Universal Robots PolyScope program: UR_con_pick.urp

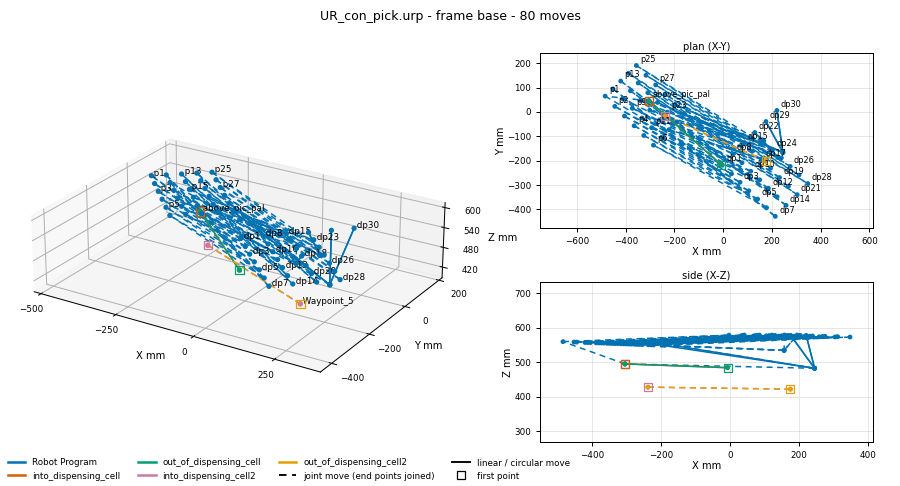
[picture p0: tool path of UR_con_pick.urp in frame base, 80 of 84 moves have a stored position in this frame; points joined in program order, loops and branches not executed]
Program UR_con_pick (installation=koniku1 directory=/programs/usbdisk createdIn=5.8.2.10297 lastSavedIn=5.8.2.10297 robotSerialNumber=20185300086)
Calibrated DH parameters: a=[0, -0.24355, -0.2132, 0, 0, 0]; d=[0.15185, 0, 0, 0.13105, 0.08535, 0.0921]; alpha=[1.570796, 0, 0, 1.570796, -1.570796, 0]; deltaTheta=[0, 0, 0, 0, 0, 0]
BeforeStart
  URCap Gripper Activate (Robotiq_Grippers, Robotiq Inc.) dataModel(ResetAndActivateKey=false)
  URCap Gripper (Robotiq_Grippers, Robotiq Inc.) dataModel(position=5.88235294117647, force=0.0, speed=100.0, positionInDouble=5.88235294117647, forceInDouble=0.0, speedInDouble=100.0, slaveIds=[9], blocking=true)
Robot Program (runOnlyOnce=false)
  Set DigitalOutput pin=digital_out[4]; digitalValue=0
  Set DigitalOutput pin=digital_out[5]; digitalValue=0
  Set DigitalOutput pin=digital_out[6]; digitalValue=1
  Wait DigitalInput pin=digital_in[0]; digitalValue=1
  Wait Sleep waitTime=2
  Set DigitalOutput pin=digital_out[4]; digitalValue=1
  SuppressedNode
    Call into_dispensing_cell
  Set DigitalOutput pin=digital_out[6]; digitalValue=0
  SuppressedNode
    Wait Sleep waitTime=4
  SuppressedNode
    Set DigitalOutput pin=digital_out[4]; digitalValue=0
  SuppressedNode
    Call out_of_dispensing_cell
  SuppressedNode
    URCap Palletizing (pallet-impl, Universal Robots) dataModel(palletFeature=Base, isPalletizing=true, Variable(key=globalCountingVariable, variable(name=Pallet_1_cnt, initializeExpression=1)), Variable(key=layerNumberVariable, variable(name=Pallet_1_lno, initializeExpression=1)), Variable(key=layerCountingVariable, variable(name=Pallet_1_lct, initializeExpression=1)), Variable(key=handleSeparatorVariable, variable(name=Pallet_1_sep, initializeExpression=False)), Variable(key=totalCountVariable, variable(name=Pallet_1_tct, initializeExpression=1)), Variable(key=name, variable(name=Pallet_pick)), Length(key=objectHeight value=0.007 unit=M), Variable(key=referencePoint, variable(featureName=referencePoint)), Variable(key=separatorPoint, variable(featureName=separatorPoint))); state(isChildrenLocked=true)
      URCap Patterns (pallet-impl, Universal Robots) state(isChildrenLocked=true)
        URCap Pattern (pallet-impl, Universal Robots) dataModel(UUID=97f9e36b-b9de-4589-9d53-87cbb1149383, patternType=GRID, rows=6, columns=5, Variable(key=nameVariable, variable(name=Grid_Pattern_1))); state(isChildrenLocked=true)
          URCap Item (pallet-impl, Universal Robots) dataModel(UUID=9fdc5ce5-b6e0-4f8b-9b1e-b639d3105400, patternType=GRID, index=0, calibrationDeltaTheta=[0.0, 0.0, 0.0, 0.0, 0.0, 0.0], calibrationA=[0.0, -0.24355, -0.2132, 0.0, 0.0, 0.0], calibrationD=[0.15185, 0.0, 0.0, 0.13105, 0.08535, 0.0921], calibrationAlpha=[1.570796327, 0.0, 0.0, 1.570796327, -1.570796327, 0.0], calibrationJointChecksum=[-1525335148, -1523615429, 619026048, -1531415990, -1531167408, -1531364241], calibrationStatus=0, calibrationValidChecksum=true, baseToFeature=[0.0, 0.0, 0.0, 0.0, 0.0, 0.0], TCPOffset=[-6.894368318605126E-7, -2.07012625763614E-7, 0.1333485508551246, -1.2879135567015372E-5, -3.579099897030376E-5, -5.053468869036781E-5], Variable(key=variable, variable(name=CornerItem_1)), JointPositions(key=jointpositions, JointPosition(key=[1], Angle(key=pos value=-2.044884 unit=RAD)), JointPosition(key=[2], Angle(key=pos value=-0.856007 unit=RAD)), JointPosition(key=[3], Angle(key=pos value=-2.403818 unit=RAD)), JointPosition(key=[4], Angle(key=pos value=4.830618 unit=RAD)), JointPosition(key=[5], Angle(key=pos value=-1.570796 unit=RAD)), JointPosition(key=[6], Angle(key=pos value=-16.054292 unit=RAD))))
          URCap Item (pallet-impl, Universal Robots) dataModel(UUID=f3709c4d-76ab-41cc-a6c5-38be900e9d84, patternType=GRID, index=1, calibrationDeltaTheta=[0.0, 0.0, 0.0, 0.0, 0.0, 0.0], calibrationA=[0.0, -0.24355, -0.2132, 0.0, 0.0, 0.0], calibrationD=[0.15185, 0.0, 0.0, 0.13105, 0.08535, 0.0921], calibrationAlpha=[1.570796327, 0.0, 0.0, 1.570796327, -1.570796327, 0.0], calibrationJointChecksum=[-1525335148, -1523615429, 619026048, -1531415990, -1531167408, -1531364241], calibrationStatus=0, calibrationValidChecksum=true, baseToFeature=[0.0, 0.0, 0.0, 0.0, 0.0, 0.0], TCPOffset=[9.229372619434795E-6, 4.396498844233543E-6, 0.13334323666807257, 8.477001825635972E-7, 1.327940618171235E-5, -6.189188592309372E-6], Variable(key=variable, variable(name=CornerItem_2)), JointPositions(key=jointpositions, JointPosition(key=[1], Angle(key=pos value=-3.207338 unit=RAD)), JointPosition(key=[2], Angle(key=pos value=-2.009976 unit=RAD)), JointPosition(key=[3], Angle(key=pos value=-1.425001 unit=RAD)), JointPosition(key=[4], Angle(key=pos value=5.005772 unit=RAD)), JointPosition(key=[5], Angle(key=pos value=-1.570799 unit=RAD)), JointPosition(key=[6], Angle(key=pos value=-14.891838 unit=RAD))))
          URCap Item (pallet-impl, Universal Robots) dataModel(UUID=b1ca3af2-4687-467f-91fb-343ff1b58222, patternType=GRID, index=2, calibrationDeltaTheta=[0.0, 0.0, 0.0, 0.0, 0.0, 0.0], calibrationA=[0.0, -0.24355, -0.2132, 0.0, 0.0, 0.0], calibrationD=[0.15185, 0.0, 0.0, 0.13105, 0.08535, 0.0921], calibrationAlpha=[1.570796327, 0.0, 0.0, 1.570796327, -1.570796327, 0.0], calibrationJointChecksum=[-1525335148, -1523615429, 619026048, -1531415990, -1531167408, -1531364241], calibrationStatus=0, calibrationValidChecksum=true, baseToFeature=[0.0, 0.0, 0.0, 0.0, 0.0, 0.0], TCPOffset=[-9.4082809781737E-7, -6.116791892427087E-6, 0.13334862076342463, -6.130929521330413E-6, 5.636271222705123E-6, -2.025583096883148E-5], Variable(key=variable, variable(name=CornerItem_3)), JointPositions(key=jointpositions, JointPosition(key=[1], Angle(key=pos value=-3.369578 unit=RAD)), JointPosition(key=[2], Angle(key=pos value=-1.900962 unit=RAD)), JointPosition(key=[3], Angle(key=pos value=-1.583163 unit=RAD)), JointPosition(key=[4], Angle(key=pos value=5.05492 unit=RAD)), JointPosition(key=[5], Angle(key=pos value=-1.570799 unit=RAD)), JointPosition(key=[6], Angle(key=pos value=-14.729598 unit=RAD))))
          URCap Item (pallet-impl, Universal Robots) dataModel(UUID=ef6c2500-fb10-456a-befd-b56711e1c953, patternType=GRID, index=3, calibrationDeltaTheta=[0.0, 0.0, 0.0, 0.0, 0.0, 0.0], calibrationA=[0.0, -0.24355, -0.2132, 0.0, 0.0, 0.0], calibrationD=[0.15185, 0.0, 0.0, 0.13105, 0.08535, 0.0921], calibrationAlpha=[1.570796327, 0.0, 0.0, 1.570796327, -1.570796327, 0.0], calibrationJointChecksum=[-1525335148, -1523615429, 619026048, -1531415990, -1531167408, -1531364241], calibrationStatus=0, calibrationValidChecksum=true, baseToFeature=[0.0, 0.0, 0.0, 0.0, 0.0, 0.0], TCPOffset=[2.1432504664631313E-6, -6.584905607454061E-7, 0.13334782612851442, -1.4261198173061594E-5, -2.9604863100931024E-6, -1.620282006412827E-5], Variable(key=variable, variable(name=CornerItem_4)), JointPositions(key=jointpositions, JointPosition(key=[1], Angle(key=pos value=-1.784534 unit=RAD)), JointPosition(key=[2], Angle(key=pos value=-0.178707 unit=RAD)), JointPosition(key=[3], Angle(key=pos value=-2.390402 unit=RAD)), JointPosition(key=[4], Angle(key=pos value=4.139902 unit=RAD)), JointPosition(key=[5], Angle(key=pos value=-1.570795 unit=RAD)), JointPosition(key=[6], Angle(key=pos value=-16.314643 unit=RAD))))
      URCap Layers (pallet-impl, Universal Robots) dataModel(separators=[false], selectedPatterns=[97f9e36b-b9de-4589-9d53-87cbb1149383])
      URCap At Each Item (pallet-impl, Universal Robots) dataModel(currentWizardState=MANUAL, selectedPattern=97f9e36b-b9de-4589-9d53-87cbb1149383, selectedPosition=9fdc5ce5-b6e0-4f8b-9b1e-b639d3105400, Pose(key=refBaseToFeature, Position(key=posePosition, Length(key=X value=0 unit=M), Length(key=Y value=0 unit=M), Length(key=Z value=0 unit=M)), Rotation(key=poseRotation, Angle(key=RX value=0 unit=RAD), Angle(key=RY value=0 unit=RAD), Angle(key=RZ value=0 unit=RAD))), Pose(key=refPose, Position(key=posePosition, Length(key=X value=-0.343187 unit=M), Length(key=Y value=0.09747 unit=M), Length(key=Z value=0.545454 unit=M)), Rotation(key=poseRotation, Angle(key=RX value=-0.000051 unit=RAD), Angle(key=RY value=-0.000053 unit=RAD), Angle(key=RZ value=2.314257 unit=RAD))))
        URCap Generated Movements (pallet-impl, Universal Robots) state(isChildrenLocked=true)
          MoveJ speed 60 deg/s, acceleration 80 deg/s^2 (useActiveTCP=true) feature=referencePoint
            Waypoint Approach: TCP in base x=-343.176 y=97.475 z=545.47 mm, rx=0 ry=0 rz=2.3142 rad; joints [-174.305, -100.758, -98.722, 289.48, -90.001, -863.099] deg; TCP offset x=0 y=0 z=133.35 mm, rx=0 ry=0 rz=0 rad; feature pose in base x=-343.187 y=97.47 z=545.454 mm, rx=-0.0001 ry=-0.0001 rz=2.3143 rad
          MoveL speed 250 mm/s, acceleration 1200 mm/s^2 (useActiveTCP=true) feature(featureName=referencePoint)
            Waypoint ToolActionPoint: TCP in base x=-343.178 y=97.469 z=568.911 mm, rx=0 ry=-0.0001 rz=2.3142 rad; joints [-174.305, -99.195, -94.039, 283.232, -90.002, -863.1] deg
          Folder Tool action
            URCap Gripper (Robotiq_Grippers, Robotiq Inc.) dataModel(position=100.0, force=100.0, speed=100.0, positionInDouble=100.0, forceInDouble=100.0, speedInDouble=100.0, slaveIds=[9], blocking=true)
          MoveL speed 250 mm/s, acceleration 1200 mm/s^2 (useActiveTCP=true) feature(featureName=referencePoint)
            Waypoint Exit_1: TCP in base x=-343.172 y=97.481 z=545.474 mm, rx=0 ry=0 rz=2.3142 rad; joints [-174.305, -100.758, -98.722, 289.48, -90, -863.099] deg
  MoveJ speed 60 deg/s, acceleration 80 deg/s^2 (useActiveTCP=true positionType=JointAngles) feature=Base
    Waypoint above_pic_pal: motionParameters(blendRadius=0.05); TCP in base x=-304.693 y=45.552 z=495.693 mm, rx=0.0433 ry=0.0193 rz=2.3479 rad; joints [-32.715, -82.821, 118.956, -127.904, 91.195, -1182.761] deg; feature pose in base x=-497.069 y=75.993 z=579.86 mm, rx=-2.8904 ry=-1.1945 rz=0.0548 rad
  MoveJ speed 60 deg/s, acceleration 80 deg/s^2 (useActiveTCP=true positionType=JointAngles) feature=pic_pallet
    Waypoint p1: TCP in base x=-484.557 y=64.859 z=560.272 mm, rx=0.0433 ry=0.0194 rz=2.3475 rad; joints [-22.755, -41.69, 36.782, -87.039, 90.875, -1192.739] deg; feature pose in base x=-497.069 y=75.993 z=579.86 mm, rx=-2.8904 ry=-1.1945 rz=0.0548 rad
    Call pic
    Call into_dispensing_cell
    MoveJ speed 60 deg/s, acceleration 80 deg/s^2 (useActiveTCP=true positionType=JointAngles) feature=disp_pallet
      Waypoint dp1: TCP in base x=-3.424 y=-217.799 z=579.158 mm, rx=-0.0069 ry=0.0195 rz=-2.3497 rad; joints [50.912, -121.659, 123.059, -91.26, 89.08, -1175.545] deg; feature pose in base x=-22.765 y=-224.486 z=598.706 mm, rx=-2.8794 ry=-1.2177 rz=0.0087 rad
    Call place
    Call out_of_dispensing_cell
    Waypoint p2: TCP in base x=-444.833 y=22.81 z=558.891 mm, rx=0.0435 ry=0.0194 rz=2.3477 rad; joints [-19.64, -55.719, 61.77, -98.051, 90.767, -1195.84] deg; feature pose in base x=-497.069 y=75.993 z=579.86 mm, rx=-2.8904 ry=-1.1945 rz=0.0548 rad
    Call pic
    Call into_dispensing_cell
    MoveJ speed 60 deg/s, acceleration 80 deg/s^2 (useActiveTCP=true positionType=JointAngles) feature=disp_pallet
      Waypoint dp2: TCP in base x=34.254 y=-254.321 z=578.313 mm, rx=-0.0002 ry=-0.0007 rz=-2.3499 rad; joints [66.977, -108.075, 116.317, -98.272, 90.015, -1191.614] deg; feature pose in base x=-22.765 y=-224.486 z=598.706 mm, rx=-2.8794 ry=-1.2177 rz=0.0087 rad
    Call place
    Call out_of_dispensing_cell
    Waypoint p3: TCP in base x=-405.137 y=-17.016 z=557.432 mm, rx=0.0435 ry=0.0195 rz=2.3477 rad; joints [-16.072, -66.014, 78.274, -104.307, 90.645, -1199.405] deg; feature pose in base x=-497.069 y=75.993 z=579.86 mm, rx=-2.8904 ry=-1.1945 rz=0.0548 rad
    Call pic
    Call into_dispensing_cell
    MoveJ speed 60 deg/s, acceleration 80 deg/s^2 (useActiveTCP=true positionType=JointAngles) feature=disp_pallet
      Waypoint dp3: TCP in base x=69.39 y=-288.804 z=577.487 mm, rx=-0.0072 ry=0.0194 rz=-2.3498 rad; joints [76.671, -97.472, 108.422, -100.432, 89.224, -1201.31] deg; TCP offset x=0 y=0 z=133.35 mm, rx=0 ry=0 rz=0 rad; feature pose in base x=-22.765 y=-224.486 z=598.706 mm, rx=-2.8794 ry=-1.2177 rz=0.0087 rad
    Call place
    Call out_of_dispensing_cell
    Waypoint p4: TCP in base x=-365.486 y=-56.836 z=556.01 mm, rx=0.0434 ry=0.0194 rz=2.3477 rad; joints [-11.598, -74.608, 90.688, -108.164, 90.482, -1203.876] deg; TCP offset x=0 y=0 z=133.35 mm, rx=0 ry=0 rz=0 rad; feature pose in base x=-497.069 y=75.993 z=579.86 mm, rx=-2.8904 ry=-1.1945 rz=0.0548 rad
    Call pic
    Call into_dispensing_cell
    MoveJ speed 60 deg/s, acceleration 80 deg/s^2 (useActiveTCP=true positionType=JointAngles) feature=disp_pallet
      Waypoint dp4: TCP in base x=105.198 y=-323.736 z=577.111 mm, rx=0.0002 ry=-0.0003 rz=-2.3344 rad; joints [85.369, -85.285, 96.899, -101.619, 90.015, -1209.121] deg; feature pose in base x=-22.765 y=-224.486 z=598.706 mm, rx=-2.8794 ry=-1.2177 rz=0.0087 rad
    Call place
    Call out_of_dispensing_cell
    Waypoint p5: TCP in base x=-325.801 y=-96.685 z=554.556 mm, rx=0.0433 ry=0.0195 rz=2.3478 rad; joints [-5.955, -81.831, 100.097, -110.387, 90.276, -1209.511] deg; feature pose in base x=-497.069 y=75.993 z=579.86 mm, rx=-2.8904 ry=-1.1945 rz=0.0548 rad
    Call pic
    Call into_dispensing_cell
    MoveJ speed 60 deg/s, acceleration 80 deg/s^2 (useActiveTCP=true positionType=JointAngles) feature=disp_pallet
      Waypoint dp5: TCP in base x=141.536 y=-357.763 z=576.271 mm, rx=-0.007 ry=0.0194 rz=-2.334 rad; joints [91.282, -75.126, 84.672, -98.851, 89.379, -1215.017] deg; feature pose in base x=-22.765 y=-224.486 z=598.706 mm, rx=-2.8794 ry=-1.2177 rz=0.0087 rad
    Call place
    Call out_of_dispensing_cell
    Waypoint p6: TCP in base x=-286.125 y=-136.528 z=553.087 mm, rx=0.0434 ry=0.0194 rz=2.3478 rad; joints [1.099, -87.499, 106.825, -111.465, 90.009, -1216.562] deg; feature pose in base x=-497.069 y=75.993 z=579.86 mm, rx=-2.8904 ry=-1.1945 rz=0.0548 rad
    Call pic
    Call into_dispensing_cell
    MoveJ speed 60 deg/s, acceleration 80 deg/s^2 (useActiveTCP=true positionType=JointAngles) feature=disp_pallet
      Waypoint dp6: TCP in base x=177.906 y=-393.046 z=575.438 mm, rx=-0.007 ry=0.0196 rz=-2.34 rad; joints [96.365, -63.254, 68.151, -94.14, 89.444, -1220.444] deg; feature pose in base x=-22.765 y=-224.486 z=598.706 mm, rx=-2.8794 ry=-1.2177 rz=0.0087 rad
    Call place
    Call out_of_dispensing_cell
    Waypoint p7: TCP in base x=-452.507 y=94.589 z=559.158 mm, rx=0.0434 ry=0.0194 rz=2.3477 rad; joints [-27.746, -50.904, 53.535, -94.5, 91.042, -1187.739] deg; feature pose in base x=-497.069 y=75.993 z=579.86 mm, rx=-2.8904 ry=-1.1945 rz=0.0548 rad
    Call pic
    Call into_dispensing_cell
    MoveJ speed 60 deg/s, acceleration 80 deg/s^2 (useActiveTCP=true positionType=JointAngles) feature=disp_pallet
      Waypoint dp7: TCP in base x=213.97 y=-428.647 z=574.564 mm, rx=-0.0071 ry=0.0196 rz=-2.3477 rad; joints [100.408, -49.228, 45.455, -85.434, 89.501, -1224.927] deg; feature pose in base x=-22.765 y=-224.486 z=598.706 mm, rx=-2.8794 ry=-1.2177 rz=0.0087 rad
    Call place
    Call out_of_dispensing_cell
    Waypoint p8: TCP in base x=-412.822 y=54.737 z=557.688 mm, rx=0.0434 ry=0.0195 rz=2.3477 rad; joints [-25.345, -63.333, 74.131, -102.709, 90.967, -1190.138] deg; feature pose in base x=-497.069 y=75.993 z=579.86 mm, rx=-2.8904 ry=-1.1945 rz=0.0548 rad
    Call pic
    Call into_dispensing_cell
    MoveJ speed 60 deg/s, acceleration 80 deg/s^2 (useActiveTCP=true positionType=JointAngles) feature=disp_pallet
      Waypoint dp8: TCP in base x=40.978 y=-172.989 z=579.404 mm, rx=0.0183 ry=-0.0109 rz=-2.3354 rad; joints [57.452, -135.568, 126.871, -80.897, 90.874, -1181.26] deg; feature pose in base x=-22.765 y=-224.486 z=598.706 mm, rx=-2.8794 ry=-1.2177 rz=0.0087 rad
    Call place
    Call out_of_dispensing_cell
    Waypoint p9: TCP in base x=-373.12 y=14.889 z=556.24 mm, rx=0.0435 ry=0.0195 rz=2.3477 rad; joints [-22.276, -73.765, 89.457, -107.657, 90.861, -1193.209] deg; feature pose in base x=-497.069 y=75.993 z=579.86 mm, rx=-2.8904 ry=-1.1945 rz=0.0548 rad
    Call pic
    Call into_dispensing_cell
    MoveJ speed 60 deg/s, acceleration 80 deg/s^2 (useActiveTCP=true positionType=JointAngles) feature=disp_pallet
      Waypoint dp9: TCP in base x=77.279 y=-208.523 z=578.499 mm, rx=0.0001 ry=-0.0005 rz=-2.3497 rad; joints [74.248, -119.104, 122.229, -93.14, 90.016, -1198.878] deg; TCP offset x=0 y=0 z=133.35 mm, rx=0 ry=0 rz=0 rad; feature pose in base x=-22.765 y=-224.486 z=598.706 mm, rx=-2.8794 ry=-1.2177 rz=0.0087 rad
    Call place
    Call out_of_dispensing_cell
    Waypoint p10: TCP in base x=-333.429 y=-24.957 z=554.774 mm, rx=0.0435 ry=0.0195 rz=2.3477 rad; joints [-18.266, -83.133, 101.5, -110.388, 90.723, -1197.216] deg; TCP offset x=0 y=0 z=133.35 mm, rx=0 ry=0 rz=0 rad; feature pose in base x=-497.069 y=75.993 z=579.86 mm, rx=-2.8904 ry=-1.1945 rz=0.0548 rad
    Call pic
    Call into_dispensing_cell
    MoveJ speed 60 deg/s, acceleration 80 deg/s^2 (useActiveTCP=true positionType=JointAngles) feature=disp_pallet
      Waypoint dp10: TCP in base x=113.244 y=-243.464 z=577.675 mm, rx=0.0001 ry=-0.0005 rz=-2.3498 rad; joints [85.746, -104.536, 114.095, -99.576, 90.015, -1210.382] deg; TCP offset x=0 y=0 z=133.35 mm, rx=0 ry=0 rz=0 rad; feature pose in base x=-22.765 y=-224.486 z=598.706 mm, rx=-2.8794 ry=-1.2177 rz=0.0087 rad
    Call place
    Call out_of_dispensing_cell
    Waypoint p11: TCP in base x=-293.737 y=-64.804 z=553.329 mm, rx=0.0436 ry=0.0195 rz=2.3476 rad; joints [-12.944, -91.552, 110.826, -111.357, 90.533, -1202.537] deg; TCP offset x=0 y=0 z=133.35 mm, rx=0 ry=0 rz=0 rad; feature pose in base x=-497.069 y=75.993 z=579.86 mm, rx=-2.8904 ry=-1.1945 rz=0.0548 rad
    Call pic
    Call into_dispensing_cell
    MoveJ speed 60 deg/s, acceleration 80 deg/s^2 (useActiveTCP=true positionType=JointAngles) feature=disp_pallet
      Waypoint dp11: TCP in base x=149.559 y=-278.719 z=577.192 mm, rx=0 ry=-0.0004 rz=-2.3499 rad; joints [93.748, -91.43, 103.232, -101.819, 90.008, -1218.386] deg; TCP offset x=0 y=0 z=133.35 mm, rx=0 ry=0 rz=0 rad; feature pose in base x=-22.765 y=-224.486 z=598.706 mm, rx=-2.8794 ry=-1.2177 rz=0.0087 rad
    Call place
    Call out_of_dispensing_cell
    Waypoint p12: TCP in base x=-254.061 y=-104.634 z=551.867 mm, rx=0.0435 ry=0.0196 rz=2.3477 rad; joints [-5.846, -98.61, 117.566, -111.087, 90.275, -1209.629] deg; TCP offset x=0 y=0 z=133.35 mm, rx=0 ry=0 rz=0 rad; feature pose in base x=-497.069 y=75.993 z=579.86 mm, rx=-2.8904 ry=-1.1945 rz=0.0548 rad
    Call pic
    Call into_dispensing_cell
    MoveJ speed 60 deg/s, acceleration 80 deg/s^2 (useActiveTCP=true positionType=JointAngles) feature=disp_pallet
      Waypoint dp12: TCP in base x=185.689 y=-313.496 z=576.033 mm, rx=0.0001 ry=-0.0004 rz=-2.3499 rad; joints [99.564, -79.257, 90.227, -100.987, 90.007, -1224.205] deg; TCP offset x=0 y=0 z=133.35 mm, rx=0 ry=0 rz=0 rad; feature pose in base x=-22.765 y=-224.486 z=598.706 mm, rx=-2.8794 ry=-1.2177 rz=0.0087 rad
    Call place
    Call out_of_dispensing_cell
    Waypoint p13: TCP in base x=-420.496 y=126.524 z=557.919 mm, rx=0.0433 ry=0.0194 rz=2.3477 rad; joints [-33.454, -57.538, 64.904, -99.118, 91.221, -1182.033] deg; TCP offset x=0 y=0 z=133.35 mm, rx=0 ry=0 rz=0 rad; feature pose in base x=-497.069 y=75.993 z=579.86 mm, rx=-2.8904 ry=-1.1945 rz=0.0548 rad
    Call pic
    Call into_dispensing_cell
    MoveJ speed 60 deg/s, acceleration 80 deg/s^2 (useActiveTCP=true positionType=JointAngles) feature=disp_pallet
      Waypoint dp13: TCP in base x=221.568 y=-348.223 z=575.153 mm, rx=0.0001 ry=-0.0004 rz=-2.35 rad; joints [103.959, -67.151, 74.321, -97.186, 90.007, -1228.606] deg; TCP offset x=0 y=0 z=133.35 mm, rx=0 ry=0 rz=0 rad; feature pose in base x=-22.765 y=-224.486 z=598.706 mm, rx=-2.8794 ry=-1.2177 rz=0.0087 rad
    Call place
    Call out_of_dispensing_cell
    Waypoint p14: TCP in base x=-380.809 y=86.65 z=556.462 mm, rx=0.0434 ry=0.0193 rz=2.3478 rad; joints [-31.714, -69.716, 83.778, -105.854, 91.163, -1183.768] deg; TCP offset x=0 y=0 z=133.35 mm, rx=0 ry=0 rz=0 rad; feature pose in base x=-497.069 y=75.993 z=579.86 mm, rx=-2.8904 ry=-1.1945 rz=0.0548 rad
    Call pic
    Call into_dispensing_cell
    MoveJ speed 60 deg/s, acceleration 80 deg/s^2 (useActiveTCP=true positionType=JointAngles) feature=disp_pallet
      Waypoint dp14: TCP in base x=258.197 y=-383.238 z=574.245 mm, rx=0.0001 ry=-0.0004 rz=-2.3501 rad; joints [107.498, -53.559, 53.294, -89.754, 90.008, -1232.146] deg; TCP offset x=0 y=0 z=133.35 mm, rx=0 ry=0 rz=0 rad; feature pose in base x=-22.765 y=-224.486 z=598.706 mm, rx=-2.8794 ry=-1.2177 rz=0.0087 rad
    Call place
    Call out_of_dispensing_cell
    Waypoint p15: TCP in base x=-341.121 y=46.802 z=555.013 mm, rx=0.0434 ry=0.0193 rz=2.3478 rad; joints [-29.413, -80.761, 98.586, -109.665, 91.091, -1186.065] deg; TCP offset x=0 y=0 z=133.35 mm, rx=0 ry=0 rz=0 rad; feature pose in base x=-497.069 y=75.993 z=579.86 mm, rx=-2.8904 ry=-1.1945 rz=0.0548 rad
    Call pic
    Call into_dispensing_cell2
    MoveJ speed 60 deg/s, acceleration 80 deg/s^2 (useActiveTCP=true positionType=JointAngles) feature=disp_pallet
      Waypoint dp15: TCP in base x=85.036 y=-125.765 z=579.34 mm, rx=0.0056 ry=0.0245 rz=0.7963 rad; joints [3.276, -178.842, 112.616, -25.169, 90.161, -1307.651] deg; TCP offset x=0 y=0 z=133.35 mm, rx=0 ry=0 rz=0 rad; feature pose in base x=-22.765 y=-224.486 z=598.706 mm, rx=-2.8794 ry=-1.2177 rz=0.0087 rad
    Call place
    Call out_of_dispensing_cell2
    Waypoint p16: TCP in base x=-301.439 y=6.972 z=553.549 mm, rx=0.0434 ry=0.0193 rz=2.3478 rad; joints [-26.269, -91.381, 110.519, -111.034, 90.989, -1189.211] deg; TCP offset x=0 y=0 z=133.35 mm, rx=0 ry=0 rz=0 rad; feature pose in base x=-497.069 y=75.993 z=579.86 mm, rx=-2.8904 ry=-1.1945 rz=0.0548 rad
    Call pic
    Call into_dispensing_cell2
    MoveJ speed 60 deg/s, acceleration 80 deg/s^2 (useActiveTCP=true positionType=JointAngles) feature=disp_pallet
      Waypoint dp16: TCP in base x=121.217 y=-160.421 z=579.288 mm, rx=0.0057 ry=0.0245 rz=0.7963 rad; joints [-13.05, -183.035, 95.361, -3.619, 90.545, -1291.327] deg; TCP offset x=0 y=0 z=133.35 mm, rx=0 ry=0 rz=0 rad; feature pose in base x=-22.765 y=-224.486 z=598.706 mm, rx=-2.8794 ry=-1.2177 rz=0.0087 rad
    Call place
    Call out_of_dispensing_cell2
    Waypoint p17: TCP in base x=-261.762 y=-32.874 z=552.083 mm, rx=0.0433 ry=0.0194 rz=2.3479 rad; joints [-21.803, -101.681, 119.854, -110.138, 90.84, -1193.669] deg; TCP offset x=0 y=0 z=133.35 mm, rx=0 ry=0 rz=0 rad; feature pose in base x=-497.069 y=75.993 z=579.86 mm, rx=-2.8904 ry=-1.1945 rz=0.0548 rad
    Call pic
    Call into_dispensing_cell2
    MoveJ speed 60 deg/s, acceleration 80 deg/s^2 (useActiveTCP=true positionType=JointAngles) feature=disp_pallet
      Waypoint dp17: TCP in base x=157.656 y=-195.07 z=579.55 mm, rx=0.0057 ry=0.0245 rz=0.7964 rad; joints [-20.295, -181.436, 77.151, 13.069, 90.704, -1284.078] deg; TCP offset x=0 y=0 z=133.35 mm, rx=0 ry=0 rz=0 rad; feature pose in base x=-22.765 y=-224.486 z=598.706 mm, rx=-2.8794 ry=-1.2177 rz=0.0087 rad
    Call place
    MoveJ speed 60 deg/s, acceleration 80 deg/s^2 (useActiveTCP=true) feature=Base
      Waypoint Waypoint_7: TCP in base x=156.47 y=-193.864 z=534.97 mm, rx=0.0058 ry=0.0246 rz=0.7964 rad; joints [-20.095, -191.819, 86.679, 13.917, 90.698, -1284.278] deg; TCP offset x=0 y=0 z=133.35 mm, rx=0 ry=0 rz=0 rad
    Call out_of_dispensing_cell2
    Waypoint p18: TCP in base x=-222.073 y=-72.72 z=550.63 mm, rx=0.0434 ry=0.0194 rz=2.3479 rad; joints [-15.273, -111.095, 126.544, -107.498, 90.61, -1200.194] deg; feature pose in base x=-497.069 y=75.993 z=579.86 mm, rx=-2.8904 ry=-1.1945 rz=0.0548 rad
    Call pic
    Call into_dispensing_cell2
    MoveJ speed 60 deg/s, acceleration 80 deg/s^2 (useActiveTCP=true) feature=Base
      Waypoint Waypoint_7: TCP in base x=156.47 y=-193.864 z=534.97 mm, rx=0.0058 ry=0.0246 rz=0.7964 rad; joints [-20.095, -191.819, 86.679, 13.917, 90.698, -1284.278] deg
    MoveJ speed 60 deg/s, acceleration 80 deg/s^2 (useActiveTCP=true positionType=JointAngles) feature=disp_pallet
      Waypoint dp18: TCP in base x=194.431 y=-230.663 z=579.465 mm, rx=0.0056 ry=0.0245 rz=0.7964 rad; joints [-24.785, -175.622, 54.194, 30.273, 90.799, -1279.589] deg; TCP offset x=0 y=0 z=133.35 mm, rx=0 ry=0 rz=0 rad; feature pose in base x=-22.765 y=-224.486 z=598.706 mm, rx=-2.8794 ry=-1.2177 rz=0.0087 rad
    Call place
    MoveJ speed 60 deg/s, acceleration 80 deg/s^2 (useActiveTCP=true) feature=Base
      Waypoint Waypoint_7: TCP in base x=156.47 y=-193.864 z=534.97 mm, rx=0.0058 ry=0.0246 rz=0.7964 rad; joints [-20.095, -191.819, 86.679, 13.917, 90.698, -1284.278] deg; TCP offset x=0 y=0 z=133.35 mm, rx=0 ry=0 rz=0 rad
    Call out_of_dispensing_cell2
    Waypoint p19: TCP in base x=-388.47 y=158.483 z=556.681 mm, rx=0.0433 ry=0.0195 rz=2.3477 rad; joints [-39.603, -62.676, 73.281, -102.215, 91.404, -1175.886] deg; feature pose in base x=-497.069 y=75.993 z=579.86 mm, rx=-2.8904 ry=-1.1945 rz=0.0548 rad
    Call pic
    Call into_dispensing_cell
    MoveJ speed 60 deg/s, acceleration 80 deg/s^2 (useActiveTCP=true positionType=JointAngles) feature=disp_pallet
      Waypoint dp19: TCP in base x=231.039 y=-269.369 z=575.995 mm, rx=0.0001 ry=-0.0004 rz=-2.3499 rad; joints [108.951, -81.607, 93.043, -101.453, 90.004, -1233.593] deg; feature pose in base x=-22.765 y=-224.486 z=598.706 mm, rx=-2.8794 ry=-1.2177 rz=0.0087 rad
    Call place
    Call out_of_dispensing_cell
    Waypoint p20: TCP in base x=-348.764 y=118.633 z=555.243 mm, rx=0.0433 ry=0.0194 rz=2.3476 rad; joints [-38.725, -75.072, 91.323, -107.887, 91.379, -1176.765] deg; feature pose in base x=-497.069 y=75.993 z=579.86 mm, rx=-2.8904 ry=-1.1945 rz=0.0548 rad
    Call pic
    Call into_dispensing_cell
    MoveJ speed 60 deg/s, acceleration 80 deg/s^2 (useActiveTCP=true positionType=JointAngles) feature=disp_pallet
      Waypoint dp20: TCP in base x=267.664 y=-304.41 z=575.134 mm, rx=0 ry=-0.0004 rz=-2.35 rad; joints [112.463, -69.027, 77.009, -98.002, 90.002, -1237.108] deg; feature pose in base x=-22.765 y=-224.486 z=598.706 mm, rx=-2.8794 ry=-1.2177 rz=0.0087 rad
    Call place
    Call out_of_dispensing_cell
    Waypoint p21: TCP in base x=-309.096 y=78.789 z=553.776 mm, rx=0.0433 ry=0.0195 rz=2.3477 rad; joints [-37.52, -87.02, 105.921, -110.563, 91.344, -1177.969] deg; feature pose in base x=-497.069 y=75.993 z=579.86 mm, rx=-2.8904 ry=-1.1945 rz=0.0548 rad
    Call pic
    Call into_dispensing_cell
    MoveJ speed 60 deg/s, acceleration 80 deg/s^2 (useActiveTCP=true positionType=JointAngles) feature=disp_pallet
      Waypoint dp21: TCP in base x=303.966 y=-339.655 z=573.762 mm, rx=0 ry=-0.0004 rz=-2.35 rad; joints [115.118, -55.451, 56.569, -91.135, 90.001, -1239.762] deg; feature pose in base x=-22.765 y=-224.486 z=598.706 mm, rx=-2.8794 ry=-1.2177 rz=0.0087 rad
    Call place
    Call out_of_dispensing_cell
    Waypoint p22: TCP in base x=-269.402 y=38.935 z=552.336 mm, rx=0.0434 ry=0.0194 rz=2.3477 rad; joints [-35.788, -99.328, 117.836, -110.213, 91.294, -1179.7] deg; feature pose in base x=-497.069 y=75.993 z=579.86 mm, rx=-2.8904 ry=-1.1945 rz=0.0548 rad
    Call pic
    Call into_dispensing_cell
    MoveL speed 250 mm/s, acceleration 1200 mm/s^2 (useActiveTCP=true) feature=disp_pallet
      Waypoint Waypoint_8: TCP in base x=224.282 y=-185.84 z=571.695 mm, rx=-0.044 ry=0.0174 rz=-2.3363 rad; joints [111.87, -99.639, 111.673, -101.289, 88, -1235.76] deg; feature pose in base x=-22.765 y=-224.486 z=598.706 mm, rx=-2.8794 ry=-1.2177 rz=0.0087 rad
      Waypoint Waypoint_9: TCP in base x=159.97 y=-114.091 z=573.27 mm, rx=-0.044 ry=0.0174 rz=-2.3363 rad; joints [99.327, -131.303, 127.646, -86.051, 87.886, -1223.211] deg
    MoveJ speed 60 deg/s, acceleration 80 deg/s^2 (useActiveTCP=true positionType=JointAngles) feature=disp_pallet
      Waypoint dp22: TCP in base x=130.171 y=-84.495 z=578.388 mm, rx=-0.0071 ry=0.0195 rz=-2.3448 rad; joints [87.55, -148.794, 127.936, -68.484, 89.335, -1211.906] deg
    Call place
    MoveL speed 250 mm/s, acceleration 1200 mm/s^2 (useActiveTCP=true) feature=disp_pallet
      Waypoint Waypoint_8: TCP in base x=224.282 y=-185.84 z=571.695 mm, rx=-0.044 ry=0.0174 rz=-2.3363 rad; joints [111.87, -99.639, 111.673, -101.289, 88, -1235.76] deg
    Call out_of_dispensing_cell
    Waypoint p23: TCP in base x=-229.733 y=-0.909 z=550.874 mm, rx=0.0434 ry=0.0194 rz=2.3477 rad; joints [-33.12, -112.367, 127.073, -106.468, 91.211, -1182.368] deg; feature pose in base x=-497.069 y=75.993 z=579.86 mm, rx=-2.8904 ry=-1.1945 rz=0.0548 rad
    Call pic
    Call into_dispensing_cell
    MoveJ speed 60 deg/s, acceleration 80 deg/s^2 (useActiveTCP=true positionType=JointAngles) feature=disp_pallet
      Waypoint dp23: TCP in base x=166.758 y=-119.289 z=578.381 mm, rx=-0.0071 ry=0.0195 rz=-2.3448 rad; joints [104.044, -126.672, 124.794, -87.304, 89.549, -1228.399] deg; feature pose in base x=-22.765 y=-224.486 z=598.706 mm, rx=-2.8794 ry=-1.2177 rz=0.0087 rad
    Call place
    Call out_of_dispensing_cell
    Waypoint p24: TCP in base x=-190.062 y=-40.733 z=549.395 mm, rx=0.0433 ry=0.0195 rz=2.3477 rad; joints [-28.635, -125.678, 133.317, -99.488, 91.072, -1186.849] deg; feature pose in base x=-497.069 y=75.993 z=579.86 mm, rx=-2.8904 ry=-1.1945 rz=0.0548 rad
    Call pic
    Call into_dispensing_cell
    MoveJ speed 60 deg/s, acceleration 80 deg/s^2 (useActiveTCP=true positionType=JointAngles) feature=disp_pallet
      Waypoint dp24: TCP in base x=203.272 y=-154.015 z=578.532 mm, rx=-0.0071 ry=0.0194 rz=-2.3448 rad; joints [111.576, -109.75, 116.936, -96.321, 89.659, -1235.93] deg; feature pose in base x=-22.765 y=-224.486 z=598.706 mm, rx=-2.8794 ry=-1.2177 rz=0.0087 rad
    Call place
    Call out_of_dispensing_cell
    Waypoint p25: TCP in base x=-356.449 y=190.438 z=555.442 mm, rx=0.0433 ry=0.0195 rz=2.3477 rad; joints [-46.108, -66.573, 79.397, -104.266, 91.577, -1169.382] deg; feature pose in base x=-497.069 y=75.993 z=579.86 mm, rx=-2.8904 ry=-1.1945 rz=0.0548 rad
    Call pic
    Call into_dispensing_cell
    MoveJ speed 60 deg/s, acceleration 80 deg/s^2 (useActiveTCP=true positionType=JointAngles) feature=disp_pallet
      Waypoint dp25: TCP in base x=238.806 y=-188.535 z=576.834 mm, rx=-0.0072 ry=0.0195 rz=-2.3449 rad; joints [115.971, -95.633, 106.852, -100.326, 89.726, -1240.329] deg; feature pose in base x=-22.765 y=-224.486 z=598.706 mm, rx=-2.8794 ry=-1.2177 rz=0.0087 rad
    Call place
    Call out_of_dispensing_cell
    Waypoint p26: TCP in base x=-316.772 y=150.578 z=554.015 mm, rx=0.0432 ry=0.0195 rz=2.3477 rad; joints [-46.273, -79.37, 97.018, -109.083, 91.581, -1169.216] deg; feature pose in base x=-497.069 y=75.993 z=579.86 mm, rx=-2.8904 ry=-1.1945 rz=0.0548 rad
    Call pic
    Call into_dispensing_cell
    MoveJ speed 60 deg/s, acceleration 80 deg/s^2 (useActiveTCP=true positionType=JointAngles) feature=disp_pallet
      Waypoint dp26: TCP in base x=275.105 y=-223.75 z=575.723 mm, rx=-0.0071 ry=0.0195 rz=-2.3448 rad; joints [119.035, -82.646, 93.938, -100.385, 89.776, -1243.39] deg; feature pose in base x=-22.765 y=-224.486 z=598.706 mm, rx=-2.8794 ry=-1.2177 rz=0.0087 rad
    Call place
    Call out_of_dispensing_cell
    Waypoint p27: TCP in base x=-277.093 y=110.747 z=552.556 mm, rx=0.0432 ry=0.0195 rz=2.3477 rad; joints [-46.508, -92.357, 111.541, -110.612, 91.588, -1168.981] deg; feature pose in base x=-497.069 y=75.993 z=579.86 mm, rx=-2.8904 ry=-1.1945 rz=0.0548 rad
    Call pic
    Call into_dispensing_cell
    MoveJ speed 60 deg/s, acceleration 80 deg/s^2 (useActiveTCP=true positionType=JointAngles) feature=disp_pallet
      Waypoint dp27: TCP in base x=311.403 y=-258.985 z=574.902 mm, rx=-0.0071 ry=0.0195 rz=-2.3448 rad; joints [121.261, -70.084, 78.17, -97.171, 89.811, -1245.615] deg; feature pose in base x=-22.765 y=-224.486 z=598.706 mm, rx=-2.8794 ry=-1.2177 rz=0.0087 rad
    Call place
    Call out_of_dispensing_cell
    Waypoint p28: TCP in base x=-237.402 y=70.897 z=551.101 mm, rx=0.0433 ry=0.0195 rz=2.3477 rad; joints [-46.864, -106.66, 123.421, -108.182, 91.597, -1168.623] deg; feature pose in base x=-497.069 y=75.993 z=579.86 mm, rx=-2.8904 ry=-1.1945 rz=0.0548 rad
    Call pic
    Call into_dispensing_cell
    MoveJ speed 60 deg/s, acceleration 80 deg/s^2 (useActiveTCP=true positionType=JointAngles) feature=disp_pallet
      Waypoint dp28: TCP in base x=347.636 y=-294.179 z=573.585 mm, rx=-0.0071 ry=0.0194 rz=-2.3449 rad; joints [122.954, -56.653, 58.204, -90.634, 89.84, -1247.31] deg; feature pose in base x=-22.765 y=-224.486 z=598.706 mm, rx=-2.8794 ry=-1.2177 rz=0.0087 rad
    Call place
    Call out_of_dispensing_cell
    Waypoint p29: TCP in base x=-197.741 y=31.055 z=549.634 mm, rx=0.0432 ry=0.0194 rz=2.3477 rad; joints [-47.467, -123.346, 132.264, -100.319, 91.609, -1168.019] deg; feature pose in base x=-497.069 y=75.993 z=579.86 mm, rx=-2.8904 ry=-1.1945 rz=0.0548 rad
    Call pic
    Call into_dispensing_cell
    MoveL speed 250 mm/s, acceleration 1200 mm/s^2 (useActiveTCP=true) feature=Base
      Waypoint Waypoint_10: TCP in base x=244.985 y=-166.148 z=483.106 mm, rx=-0.0433 ry=0.0105 rz=-2.357 rad; joints [117.959, -87.681, 127.466, -129.129, 88.108, -1243.031] deg
    MoveL speed 250 mm/s, acceleration 1200 mm/s^2 (useActiveTCP=true) feature=disp_pallet
      Waypoint dp29: TCP in base x=175.483 y=-39.366 z=578.609 mm, rx=-0.006 ry=0.0017 rz=-2.3425 rad; joints [120.102, -135.786, 127.251, -81.353, 89.74, -1244.317] deg; feature pose in base x=-22.765 y=-224.486 z=598.706 mm, rx=-2.8794 ry=-1.2177 rz=0.0087 rad
    Call place
    MoveL speed 250 mm/s, acceleration 1200 mm/s^2 (useActiveTCP=true) feature=Base
      Waypoint Waypoint_10: TCP in base x=244.985 y=-166.148 z=483.106 mm, rx=-0.0433 ry=0.0105 rz=-2.357 rad; joints [117.959, -87.681, 127.466, -129.129, 88.108, -1243.031] deg
    Call out_of_dispensing_cell
    Waypoint p30: TCP in base x=-158.044 y=-8.801 z=548.185 mm, rx=0.0433 ry=0.0194 rz=2.3478 rad; joints [-48.734, -142.94, 136.956, -85.385, 91.64, -1166.749] deg; feature pose in base x=-497.069 y=75.993 z=579.86 mm, rx=-2.8904 ry=-1.1945 rz=0.0548 rad
    Call pic
    Call into_dispensing_cell
    MoveL speed 250 mm/s, acceleration 1200 mm/s^2 (useActiveTCP=true) feature=Base
      Waypoint Waypoint_10: TCP in base x=244.985 y=-166.148 z=483.106 mm, rx=-0.0433 ry=0.0105 rz=-2.357 rad; joints [117.959, -87.681, 127.466, -129.129, 88.108, -1243.031] deg
    MoveL speed 250 mm/s, acceleration 1200 mm/s^2 (useActiveTCP=true) feature=disp_pallet
      Waypoint dp30: TCP in base x=220.533 y=6.001 z=578.391 mm, rx=-0.0061 ry=0.0018 rz=-2.3425 rad; joints [144.877, -120.134, 122.613, -92.266, 89.812, -1269.092] deg; feature pose in base x=-22.765 y=-224.486 z=598.706 mm, rx=-2.8794 ry=-1.2177 rz=0.0087 rad
    Call place
    MoveL speed 250 mm/s, acceleration 1200 mm/s^2 (useActiveTCP=true) feature=Base
      Waypoint Waypoint_10: TCP in base x=244.985 y=-166.148 z=483.106 mm, rx=-0.0433 ry=0.0105 rz=-2.357 rad; joints [117.959, -87.681, 127.466, -129.129, 88.108, -1243.031] deg
    Call out_of_dispensing_cell
    MoveJ speed 60 deg/s, acceleration 80 deg/s^2 (useActiveTCP=true positionType=JointAngles) feature=Base
      Waypoint above_pic_pal: motionParameters(blendRadius=0.05); TCP in base x=-304.693 y=45.552 z=495.693 mm, rx=0.0433 ry=0.0193 rz=2.3479 rad; joints [-32.715, -82.821, 118.956, -127.904, 91.195, -1182.761] deg; feature pose in base x=-497.069 y=75.993 z=579.86 mm, rx=-2.8904 ry=-1.1945 rz=0.0548 rad
    Halt
  SuppressedNode
    URCap Palletizing (pallet-impl, Universal Robots) dataModel(palletFeature=Base, isPalletizing=true, Variable(key=globalCountingVariable, variable(name=Pallet_2_cnt, initializeExpression=1)), Variable(key=layerNumberVariable, variable(name=Pallet_2_lno, initializeExpression=1)), Variable(key=layerCountingVariable, variable(name=Pallet_2_lct, initializeExpression=1)), Variable(key=handleSeparatorVariable, variable(name=Pallet_2_sep, initializeExpression=False)), Variable(key=totalCountVariable, variable(name=Pallet_2_tct, initializeExpression=1)), Variable(key=name, variable(name=OT_place)), Length(key=objectHeight value=0.007 unit=M), Variable(key=referencePoint, variable(featureName=referencePoin_1)), Variable(key=separatorPoint, variable(featureName=separatorPoin_1))); state(isChildrenLocked=true)
      URCap Patterns (pallet-impl, Universal Robots) state(isChildrenLocked=true)
        URCap Pattern (pallet-impl, Universal Robots) dataModel(UUID=012a3881-f614-4089-bd9a-0103003ba865, patternType=GRID, rows=6, columns=3, Variable(key=nameVariable, variable(name=Grid_Pattern_2))); state(isChildrenLocked=true)
          URCap Item (pallet-impl, Universal Robots) dataModel(UUID=b1dd0d16-fb4d-45bb-ae53-6229e1c8cc65, patternType=GRID, index=0, calibrationDeltaTheta=[0.0, 0.0, 0.0, 0.0, 0.0, 0.0], calibrationA=[0.0, -0.24355, -0.2132, 0.0, 0.0, 0.0], calibrationD=[0.15185, 0.0, 0.0, 0.13105, 0.08535, 0.0921], calibrationAlpha=[1.570796327, 0.0, 0.0, 1.570796327, -1.570796327, 0.0], calibrationJointChecksum=[-1525335148, -1523615429, 619026048, -1531415990, -1531167408, -1531364241], calibrationStatus=0, calibrationValidChecksum=true, baseToFeature=[0.0, 0.0, 0.0, 0.0, 0.0, 0.0], TCPOffset=[6.385434602740325E-7, -8.061105506440569E-7, 0.13334729456446137, -4.554708473558058E-6, 4.501659996473501E-6, -8.084013495976523E-6], Variable(key=variable, variable(name=CornerItem_5)), JointPositions(key=jointpositions, JointPosition(key=[1], Angle(key=pos value=-0.91853 unit=RAD)), JointPosition(key=[2], Angle(key=pos value=-0.967371 unit=RAD)), JointPosition(key=[3], Angle(key=pos value=-2.150649 unit=RAD)), JointPosition(key=[4], Angle(key=pos value=4.652061 unit=RAD)), JointPosition(key=[5], Angle(key=pos value=-1.576318 unit=RAD)), JointPosition(key=[6], Angle(key=pos value=-15.558283 unit=RAD))))
          URCap Item (pallet-impl, Universal Robots) dataModel(UUID=f85688ce-86fe-40be-a9aa-3f62666ac9fc, patternType=GRID, index=1, calibrationDeltaTheta=[0.0, 0.0, 0.0, 0.0, 0.0, 0.0], calibrationA=[0.0, -0.24355, -0.2132, 0.0, 0.0, 0.0], calibrationD=[0.15185, 0.0, 0.0, 0.13105, 0.08535, 0.0921], calibrationAlpha=[1.570796327, 0.0, 0.0, 1.570796327, -1.570796327, 0.0], calibrationJointChecksum=[-1525335148, -1523615429, 619026048, -1531415990, -1531167408, -1531364241], calibrationStatus=0, calibrationValidChecksum=true, baseToFeature=[0.0, 0.0, 0.0, 0.0, 0.0, 0.0], TCPOffset=[4.421324504733093E-6, -8.882263695109138E-6, 0.13335590071403947, 1.1704926281735933E-6, -1.7124720559842012E-5, -9.576729179021103E-6], Variable(key=variable, variable(name=CornerItem_6)), JointPositions(key=jointpositions, JointPosition(key=[1], Angle(key=pos value=-0.819251 unit=RAD)), JointPosition(key=[2], Angle(key=pos value=-2.230883 unit=RAD)), JointPosition(key=[3], Angle(key=pos value=-0.90148 unit=RAD)), JointPosition(key=[4], Angle(key=pos value=4.665989 unit=RAD)), JointPosition(key=[5], Angle(key=pos value=-1.572645 unit=RAD)), JointPosition(key=[6], Angle(key=pos value=-15.657507 unit=RAD))))
          URCap Item (pallet-impl, Universal Robots) dataModel(UUID=49a3a79b-a81e-4530-afce-77180ae53d82, patternType=GRID, index=2, calibrationDeltaTheta=[0.0, 0.0, 0.0, 0.0, 0.0, 0.0], calibrationA=[0.0, -0.24355, -0.2132, 0.0, 0.0, 0.0], calibrationD=[0.15185, 0.0, 0.0, 0.13105, 0.08535, 0.0921], calibrationAlpha=[1.570796327, 0.0, 0.0, 1.570796327, -1.570796327, 0.0], calibrationJointChecksum=[-1525335148, -1523615429, 619026048, -1531415990, -1531167408, -1531364241], calibrationStatus=0, calibrationValidChecksum=true, baseToFeature=[0.0, 0.0, 0.0, 0.0, 0.0, 0.0], TCPOffset=[-6.546520676092155E-6, 3.0061657615876314E-5, 0.1333210087102386, -9.05207583780044E-5, -1.9475650639820683E-5, -9.763073406628662E-6], Variable(key=variable, variable(name=CornerItem_7)), JointPositions(key=jointpositions, JointPosition(key=[1], Angle(key=pos value=-0.533168 unit=RAD)), JointPosition(key=[2], Angle(key=pos value=-2.103865 unit=RAD)), JointPosition(key=[3], Angle(key=pos value=-1.110396 unit=RAD)), JointPosition(key=[4], Angle(key=pos value=4.748875 unit=RAD)), JointPosition(key=[5], Angle(key=pos value=-1.562083 unit=RAD)), JointPosition(key=[6], Angle(key=pos value=-15.943397 unit=RAD))))
          URCap Item (pallet-impl, Universal Robots) dataModel(UUID=aeb82c55-226c-4814-8e7f-b1637aca92f5, patternType=GRID, index=3, calibrationDeltaTheta=[0.0, 0.0, 0.0, 0.0, 0.0, 0.0], calibrationA=[0.0, -0.24355, -0.2132, 0.0, 0.0, 0.0], calibrationD=[0.15185, 0.0, 0.0, 0.13105, 0.08535, 0.0921], calibrationAlpha=[1.570796327, 0.0, 0.0, 1.570796327, -1.570796327, 0.0], calibrationJointChecksum=[-1525335148, -1523615429, 619026048, -1531415990, -1531167408, -1531364241], calibrationStatus=0, calibrationValidChecksum=true, baseToFeature=[0.0, 0.0, 0.0, 0.0, 0.0, 0.0], TCPOffset=[4.267952937352798E-6, -8.267452121041297E-6, 0.13335404862525546, 3.345620117937874E-5, 1.7865608596165237E-6, -5.821796148433658E-5], Variable(key=variable, variable(name=CornerItem_8)), JointPositions(key=jointpositions, JointPosition(key=[1], Angle(key=pos value=0.215968 unit=RAD)), JointPosition(key=[2], Angle(key=pos value=-0.436388 unit=RAD)), JointPosition(key=[3], Angle(key=pos value=-2.210063 unit=RAD)), JointPosition(key=[4], Angle(key=pos value=4.196615 unit=RAD)), JointPosition(key=[5], Angle(key=pos value=-1.539712 unit=RAD)), JointPosition(key=[6], Angle(key=pos value=-16.69238 unit=RAD))))
      URCap Layers (pallet-impl, Universal Robots) dataModel(separators=[false], selectedPatterns=[012a3881-f614-4089-bd9a-0103003ba865])
      URCap At Each Item (pallet-impl, Universal Robots) dataModel(currentWizardState=MANUAL, selectedPattern=012a3881-f614-4089-bd9a-0103003ba865, selectedPosition=b1dd0d16-fb4d-45bb-ae53-6229e1c8cc65, Pose(key=refBaseToFeature, Position(key=posePosition, Length(key=X value=0 unit=M), Length(key=Y value=0 unit=M), Length(key=Z value=0 unit=M)), Rotation(key=poseRotation, Angle(key=RX value=0 unit=RAD), Angle(key=RY value=0 unit=RAD), Angle(key=RZ value=0 unit=RAD))), Pose(key=refPose, Position(key=posePosition, Length(key=X value=-0.000874 unit=M), Length(key=Y value=-0.212708 unit=M), Length(key=Z value=0.579569 unit=M)), Rotation(key=poseRotation, Angle(key=RX value=-0.018404 unit=RAD), Angle(key=RY value=0.043495 unit=RAD), Angle(key=RZ value=-2.339223 unit=RAD))))
        MoveL speed 250 mm/s, acceleration 1200 mm/s^2 (useActiveTCP=true) feature=Base
          Waypoint Waypoint_1: TCP in base x=-179.325 y=-62.438 z=486.107 mm, rx=0.0001 ry=0 rz=2.3211 rad; joints [-117.168, -54.496, -150.314, 294.81, -90.005, -919.845] deg; TCP offset x=0 y=0 z=133.35 mm, rx=0 ry=0 rz=0 rad
        URCap Generated Movements (pallet-impl, Universal Robots) state(isChildrenLocked=true)
          MoveJ speed 60 deg/s, acceleration 80 deg/s^2 (useActiveTCP=true) feature=referencePoin_1
            Waypoint Approach_1: TCP in base x=-1.693 y=-211.905 z=548.914 mm, rx=-0.0184 ry=0.0434 rz=-2.3392 rad; joints [-52.688, -55.581, -131.426, 274.904, -90.319, -891.363] deg; TCP offset x=0 y=0 z=133.35 mm, rx=0 ry=0 rz=0 rad; feature pose in base x=-0.874 y=-212.708 z=579.569 mm, rx=-0.0184 ry=0.0435 rz=-2.3392 rad
          MoveL speed 250 mm/s, acceleration 1200 mm/s^2 (useActiveTCP=true) feature(featureName=referencePoin_1)
            Waypoint ToolActionPoi_1: TCP in base x=-0.874 y=-212.708 z=579.569 mm, rx=-0.0184 ry=0.0435 rz=-2.3392 rad; joints [-52.372, -65.929, -80.964, 234.785, -90.307, -891.68] deg; TCP offset x=0 y=0 z=0 mm, rx=0 ry=0 rz=0 rad
          Folder Tool action
            URCap Gripper (Robotiq_Grippers, Robotiq Inc.) dataModel(position=0.0, force=0.0, speed=0.0, positionInDouble=0.0, forceInDouble=0.0, speedInDouble=0.0, slaveIds=[9], blocking=true)
          MoveL speed 250 mm/s, acceleration 1200 mm/s^2 (useActiveTCP=true) feature(featureName=referencePoin_1)
            Waypoint Exit_2: TCP in base x=-1.697 y=-211.912 z=548.904 mm, rx=-0.0184 ry=0.0435 rz=-2.3392 rad; joints [-52.688, -55.581, -131.428, 274.904, -90.318, -891.364] deg; TCP offset x=0 y=0 z=133.35 mm, rx=0 ry=0 rz=0 rad
  SuppressedNode
    Halt
SubProgram -> out_of_dispensing_cell2
SubProgram -> into_dispensing_cell2
SubProgram -> place
SubProgram -> pic
SubProgram -> out_of_dispensing_cell
SubProgram -> into_dispensing_cell
SubProgram into_dispensing_cell (keepSynchronizedWithDisk=false)
  MoveJ speed 60 deg/s, acceleration 80 deg/s^2 (useActiveTCP=true positionType=JointAngles) feature=pic_pallet
    Waypoint above_pic_pal: motionParameters(blendRadius=0.05); TCP in base x=-304.693 y=45.552 z=495.693 mm, rx=0.0433 ry=0.0193 rz=2.3479 rad; joints [-32.715, -82.821, 118.956, -127.904, 91.195, -1182.761] deg; feature pose in base x=-497.069 y=75.993 z=579.86 mm, rx=-2.8904 ry=-1.1945 rz=0.0548 rad
    MoveL speed 250 mm/s, acceleration 1200 mm/s^2 (useActiveTCP=true) feature=Base
      Waypoint Waypoint_3: motionParameters(blendRadius=0.05); TCP in base x=-7.413 y=-217.093 z=484.732 mm, rx=-0.044 ry=0.0175 rz=-2.3363 rad; joints [48.862, -110.616, 145.691, -126.518, 88.427, -1172.72] deg
SubProgram out_of_dispensing_cell (keepSynchronizedWithDisk=false)
  MoveL speed 250 mm/s, acceleration 1200 mm/s^2 (useActiveTCP=true) feature=Base
    Waypoint Waypoint_3: motionParameters(blendRadius=0.05); TCP in base x=-7.413 y=-217.093 z=484.732 mm, rx=-0.044 ry=0.0175 rz=-2.3363 rad; joints [48.862, -110.616, 145.691, -126.518, 88.427, -1172.72] deg
  MoveL speed 250 mm/s, acceleration 1200 mm/s^2 (useActiveTCP=true) feature=pic_pallet
    Waypoint above_pic_pal: TCP in base x=-304.693 y=45.552 z=495.693 mm, rx=0.0433 ry=0.0193 rz=2.3479 rad; joints [-32.715, -82.821, 118.956, -127.904, 91.195, -1182.761] deg; feature pose in base x=-497.069 y=75.993 z=579.86 mm, rx=-2.8904 ry=-1.1945 rz=0.0548 rad
SubProgram pic (keepSynchronizedWithDisk=false)
  MoveL speed 250 mm/s, acceleration 1200 mm/s^2 (useActiveTCP=true) feature=pic_pallet
    Waypoint approach (Relative): relativeFromPosition TCP in base x=-341.134 y=46.797 z=555.01 mm, rx=0.0434 ry=0.0193 rz=2.3478 rad; joints [-29.412, -80.76, 98.585, -109.663, 91.09, -1186.065] deg; TCP in base x=-340.575 y=46.81 z=569.989 mm, rx=0.0433 ry=0.0193 rz=2.3478 rad; joints [-29.462, -81.867, 95.704, -105.672, 91.091, -1186.014] deg
    URCap Gripper (Robotiq_Grippers, Robotiq Inc.) dataModel(position=100.0, force=0.0, speed=100.0, positionInDouble=100.0, forceInDouble=0.0, speedInDouble=100.0, slaveIds=[9], blocking=true)
    Waypoint Waypoint_2 (Relative): relativeFromPosition TCP in base x=-340.551 y=46.8 z=570.009 mm, rx=0.0434 ry=0.0193 rz=2.3479 rad; joints [-29.462, -81.869, 95.702, -105.674, 91.093, -1186.014] deg; TCP in base x=-341.138 y=46.801 z=554.994 mm, rx=0.0433 ry=0.0193 rz=2.3478 rad; joints [-29.411, -80.76, 98.588, -109.664, 91.091, -1186.065] deg
SubProgram place (keepSynchronizedWithDisk=false)
  MoveL speed 250 mm/s, acceleration 1200 mm/s^2 (useActiveTCP=true) feature=disp_pallet
    Waypoint Waypoint_4 (Relative): relativeFromPosition TCP in base x=-2.162 y=-219.006 z=579.127 mm, rx=-0.0001 ry=-0.0006 rz=-2.3498 rad; joints [52.707, -120.27, 122.567, -92.315, 90.019, -1177.341] deg; TCP in base x=-2.014 y=-219.193 z=594.118 mm, rx=-0.0001 ry=-0.0006 rz=-2.3498 rad; joints [52.785, -120.23, 118.519, -88.304, 90.021, -1177.42] deg; feature pose in base x=-22.765 y=-224.486 z=598.706 mm, rx=-2.8794 ry=-1.2177 rz=0.0087 rad
    URCap Gripper (Robotiq_Grippers, Robotiq Inc.) dataModel(position=6.0, force=0.0, speed=100.0, positionInDouble=6.0, forceInDouble=0.0, speedInDouble=100.0, slaveIds=[9], blocking=true)
    Waypoint Waypoint_31 (Relative): relativeFromPosition TCP in base x=-2.005 y=-219.182 z=594.126 mm, rx=-0.0001 ry=-0.0006 rz=-2.3499 rad; joints [52.784, -120.23, 118.518, -88.306, 90.02, -1177.421] deg; TCP in base x=-2.17 y=-219.012 z=579.114 mm, rx=-0.0001 ry=-0.0005 rz=-2.3498 rad; joints [52.706, -120.272, 122.57, -92.312, 90.019, -1177.339] deg
SubProgram into_dispensing_cell2 (keepSynchronizedWithDisk=false)
  MoveJ speed 60 deg/s, acceleration 80 deg/s^2 (useActiveTCP=true positionType=JointAngles) feature=disp_pallet
    Waypoint Waypoint_6: motionParameters(blendRadius=0.05); TCP in base x=-238.315 y=-16.697 z=428.358 mm, rx=0.0272 ry=0.0235 rz=2.5104 rad; joints [-27.909, -83.169, 147.496, -155.316, 91.207, -1178.256] deg
    Waypoint Waypoint_5: motionParameters(blendRadius=0.05); TCP in base x=174.64 y=-200.272 z=422.562 mm, rx=1.4462 ry=-0.1407 rz=2.3126 rad; joints [-19.314, -188.292, 151.795, -116.28, 89.952, -1178.279] deg
SubProgram out_of_dispensing_cell2 (keepSynchronizedWithDisk=false)
  MoveJ speed 60 deg/s, acceleration 80 deg/s^2 (useActiveTCP=true positionType=JointAngles) feature=disp_pallet
    Waypoint Waypoint_5: motionParameters(blendRadius=0.05); TCP in base x=174.64 y=-200.272 z=422.562 mm, rx=1.4462 ry=-0.1407 rz=2.3126 rad; joints [-19.314, -188.292, 151.795, -116.28, 89.952, -1178.279] deg
    Waypoint Waypoint_6: motionParameters(blendRadius=0.05); TCP in base x=-238.315 y=-16.697 z=428.358 mm, rx=0.0272 ry=0.0235 rz=2.5104 rad; joints [-27.909, -83.169, 147.496, -155.316, 91.207, -1178.256] deg
